// TIA Portal V17 export
// export: Created 2026-04-13T11:12:44.4838578Z, ExportSetting WithDefaults, DisplayName Totally Integrated Automation Portal, DisplayVersion V17 Update 4, DisplayName TIA Portal Openness, DisplayVersion V17 Update 4, DisplayName TIA Portal Version Control Interface, DisplayVersion V17, DisplayName SINAMICS Startdrive Advanced, DisplayVersion V17, DisplayName SINAMICS Startdrive G130, G150, S120, S150, SINAMICS MV, S210, DisplayVersion V17, DisplayName SINAMICS Startdrive G110M, G120, G120C, G120D, G120P, G115D, DisplayVersion V17, DisplayName STEP 7 Professional, DisplayVersion V17 Update 4, DisplayName STEP 7 Safety, DisplayVersion V17, DisplayName WinCC Professional, DisplayVersion V17 Update 4
DATA_BLOCK "B4-清洗连锁_DB"   // DB33
VERSION : 0.1
// stored: AutoNumber true, DBAccessibleFromOPCUA true, DBAccessibleFromWebserver true, InstanceOfName B4-清洗连锁, InstanceOfType FB
"B4-清洗连锁"
   // VAR
   //    TON0 : TON_TIME;
   //    TON1 : TON_TIME;
   //    TON2 { S7_SetPoint := 'True'} : TON_TIME;
   //    TON3 { S7_SetPoint := 'True'} : TON_TIME;
   //    TON4 { S7_SetPoint := 'True'} : TON_TIME;
   //    TON5 { S7_SetPoint := 'True'} : TON_TIME;
   //    TON6 { S7_SetPoint := 'True'} : TON_TIME;
   //    TON7 { S7_SetPoint := 'True'} : TON_TIME;
   //    R_TRIG { S7_SetPoint := 'True'} : Array[0..100] of R_TRIG;
   //    RT { S7_SetPoint := 'True'} : Array[0..100] of Bool;
   //    F_TRIG { S7_SetPoint := 'True'} : Array[0..100] of F_TRIG;
   //    FT { S7_SetPoint := 'True'} : Array[0..100] of Bool;
   //    BJ报警上升辅助 : Bool;
   //    BJ报警下降辅助 : Bool;
   //    BJ报警上升沿 { S7_SetPoint := 'True'} : R_TRIG;
   //    BJ报警下降沿 { S7_SetPoint := 'True'} : F_TRIG;
   //    F1 { S7_SetPoint := 'True'} : Bool;
   //    F2 : Bool;
   //    ET0 : Time;
   //    ET1 : Time;
   //    ET2 : Time;
   //    ET3 : Time;
   //    ET4 : Time;
   //    ET5 : Time;
   //    ET6 : Time;
   //    ET7 : Time;
   //    F3 : Bool;
   //    F4 : Bool;
   //    Temp_1 : Int;
   //    AERROR : Bool;
   //    t0_1s : TON_TIME;
   //    YC1 { S7_SetPoint := 'True'} : DInt;
   //    YC2 : DInt;
   //    YC3 : DInt;
   //    YC4 : DInt;
   //    YC5 : DInt;
   // END_VAR
BEGIN
END_DATA_BLOCK
